// TIA Portal V19 export
DATA_BLOCK "IO Mapping"   // DB3
{ S7_Optimized_Access := 'TRUE' }
// stored: MemoryReserve 100
   VAR
      DI : Struct
         "Safety OK" : Bool;
         "IBC Valve is Open" : Bool;
         "IBC Valve is Closed" : Bool;
         "Pump Valve is Open" : Bool;
         "Pump Valve is Closed" : Bool;
         "Flowmeter Feed Valve is Open" : Bool;
         "Flowmerter Feed Valve is Closed" : Bool;
         "Dose Valve is Open" : Bool;
         "Dose Valve is Closed" : Bool;
         "DOL Running Feedback" : Bool;
         "Spare 11" : Bool;
         "Spare 12" : Bool;
         "Spare 13" : Bool;
         "Spare 14" : Bool;
      END_STRUCT;
      DQ : Struct
         "CMD Open IBC Valve" : Bool;
         "CMD Open Pump Feed Valve" : Bool;
         "CMD Open Flowmeter Feed Valve" : Bool;
         "CMD Opend Dosing Valve" : Bool;
         "Run Motor Cooling" : Bool;
         "Spare 6" : Bool;
         "Spare 7" : Bool;
         "Spare 8" : Bool;
         "Spare 9" : Bool;
         "Spare 10" : Bool;
      END_STRUCT;
      AI : Struct
         "Line Pressure" : Int;
         "Buffer level" : Int;
         "Spare 1" : Int;
         "Spare 2" : Int;
      END_STRUCT;
   END_VAR
BEGIN
END_DATA_BLOCK
